{attribute addProperty BoxType "EL1258-0000-0016"}
{attribute addProperty Id "CtrlAT %Q*Ctrl_2D553DD113717.125"}
{attribute addProperty CRC "3715549080"}
{attribute addProperty SizeInBites "137"}
{attribute addProperty SizeInBytes "17.125"}
TYPE MTI_Outputs_Channel_DD76C798 :
STRUCT
	{attribute addProperty Name "Ctrl"}
	Ctrl AT %Q* : Ctrl_2D553DD1;
END_STRUCT
END_TYPE

(* stored: Version 1.2.0.0, ProductVersion 3.1.4024.9
   DUT MTI_Outputs_Channel_DD76C798: Id {98c3bc23-1a69-4503-b9c9-7db78054c61d} *)
